% RSLogix 500 project 6.6.RSS, saved by version 8.30.00.16 %
PROJECT "UNTITLED"    % processor: MicroLogix 1000 %

PROGRAM FILES
  LAD 2 "MAIN_PROG"  3 rungs
  LAD 3 "USER_FAULT"  1 rungs
  LAD 4 "HSC_INT"  1 rungs
  LAD 5 "STI_INT"  1 rungs
  LAD 6, 7, 8, 9, 10, 11, 12, 13, 14, 15, 16: only END

DATA FILES
  O0 OUTPUT  1 elements
  I1 INPUT  2 elements
  S2 STATUS  33 elements
  B3 BINARY  32 elements
  T4 TIMER  40 elements
  C5 COUNTER  32 elements
  R6 CONTROL  16 elements
  N7 INTEGER  105 elements

LADDER 2 "MAIN_PROG"
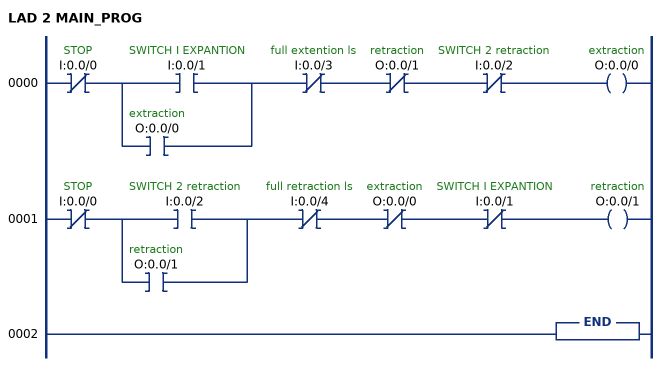
% Rung: 0 %
SOR XIO I:0.0/0 BST XIC I:0.0/1 NXB XIC O:0.0/0 BND XIO I:0.0/3 XIO O:0.0/1 XIO I:0.0/2 OTE O:0.0/0 EOR
%   I:0.0/0  "STOP" %
%   I:0.0/1  "SWITCH I EXPANTION" %
%   O:0.0/0  "extraction" %
%   I:0.0/3  "full extention ls" %
%   O:0.0/1  "retraction" %
%   I:0.0/2  "SWITCH 2 retraction" %
% Rung: 1 %
SOR XIO I:0.0/0 BST XIC I:0.0/2 NXB XIC O:0.0/1 BND XIO I:0.0/4 XIO O:0.0/0 XIO I:0.0/1 OTE O:0.0/1 EOR
%   I:0.0/0  "STOP" %
%   I:0.0/2  "SWITCH 2 retraction" %
%   O:0.0/1  "retraction" %
%   I:0.0/4  "full retraction ls" %
%   O:0.0/0  "extraction" %
%   I:0.0/1  "SWITCH I EXPANTION" %
% Rung: 2 %
SOR END EOR
